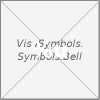
VISUALIZATION LogButton  // 100x100
VAR_IN_OUT
	nFaultsInLog : UINT;
END_VAR
    Ellipse (0,0 100x100)
    Image (0,0 100x100), image: VisuSymbols.Symbols.Bell
    Textfield (30,30 40x40), "%u", text variable: nFaultsInLog
END_VISUALIZATION

(* stored: Version 1.1.0.1, ProductVersion 3.1.4024.11
   Visu LogButton: Id {1e8540e6-ec8b-4413-918d-95dd44c3f29c} *)
